(* PLC project Unnamed, Unknown Unnamed 1 *)
(* stored: creationDateTime 2024-01-22T13:26:01, modificationDateTime 2024-01-28T15:10:34 *)

PROGRAM program0
  VAR
    FactoryIOReset AT %IX100.0 : BOOL;
    Start AT %IX100.1 : BOOL := 1;
    EmergencyStop AT %IX100.2 : BOOL;
    RetroReflect0 AT %IX100.3 : BOOL;  (* Retroreflective sensors are active low which means that the signal goes from 1 to 0 when the sensor is triggered by the pallet *)
    RetroReflect1 AT %IX100.4 : BOOL;
    RetroReflect2 AT %IX100.5 : BOOL;
    RetroReflect3 AT %IX100.6 : BOOL;
    TurntableBackLimit AT %IX100.7 : BOOL;
    TurntableFrontLimit AT %IX101.0 : BOOL;
    TurntableLimit0 AT %IX101.1 : BOOL;
    TurntableLimit90 AT %IX101.2 : BOOL;
    LightArray7 AT %IX101.3 : BOOL;
    Conveyor1 AT %QX100.0 : BOOL;
    Turntable0RollPlus AT %QX100.1 : BOOL;
    Turntable0Turn AT %QX100.2 : BOOL;
    Conveyor2 AT %QX100.3 : BOOL;
  END_VAR
  VAR
    RS0 : RS;
    RS1 : RS;
    RS2 : RS;
  END_VAR
  VAR_IN_OUT
    SmallBox : BOOL;
  END_VAR
  VAR
    RS3 : RS;
    RS4 : RS;
    RS5 : RS;
    RS6 : RS;
    RS7 : RS;
    RS8 : RS;
    RS9 : RS;
  END_VAR
  VAR  (* added by the conversion: wires and edge detectors of the diagram *)
    R_TRIG1 : R_TRIG;
    R_TRIG2 : R_TRIG;
    R_TRIG3 : R_TRIG;
    R_TRIG4 : R_TRIG;
    F_TRIG5 : F_TRIG;
    R_TRIG6 : R_TRIG;
    R_TRIG7 : R_TRIG;
    R_TRIG8 : R_TRIG;
    F_TRIG9 : F_TRIG;
    R_TRIG10 : R_TRIG;
    F_TRIG11 : F_TRIG;
    R_TRIG12 : R_TRIG;
    R_TRIG13 : R_TRIG;
    R_TRIG14 : R_TRIG;
    F_TRIG15 : F_TRIG;
    R_TRIG16 : R_TRIG;
    R_TRIG17 : R_TRIG;
    F_TRIG18 : F_TRIG;
    R_TRIG19 : R_TRIG;
    R_TRIG20 : R_TRIG;
    R_TRIG21 : R_TRIG;
    R_TRIG22 : R_TRIG;
    R_TRIG23 : R_TRIG;
    R_TRIG24 : R_TRIG;
    R_TRIG25 : R_TRIG;
  END_VAR

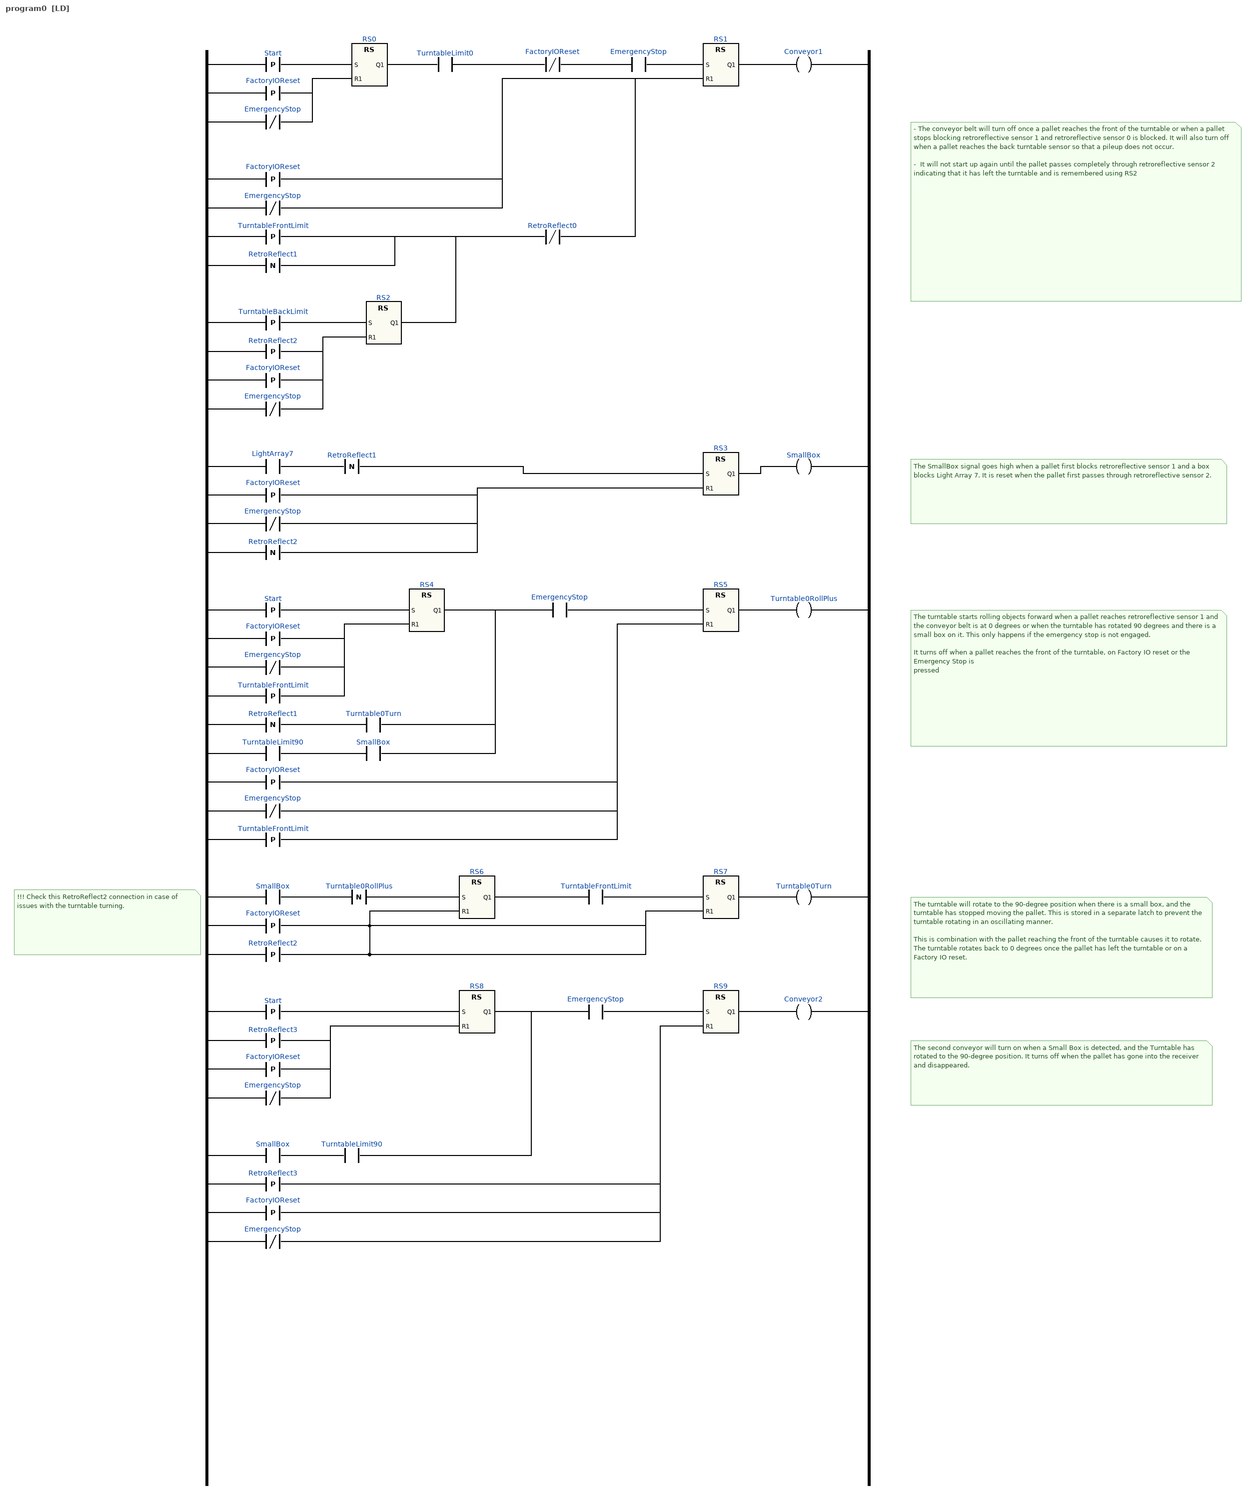
(* LD diagram, written out as Structured Text *)
R_TRIG1(CLK := Start);
R_TRIG2(CLK := FactoryIOReset);
RS0(S := R_TRIG1.Q, R1 := R_TRIG2.Q OR NOT EmergencyStop);
R_TRIG3(CLK := FactoryIOReset);
R_TRIG4(CLK := TurntableFrontLimit);
F_TRIG5(CLK := RetroReflect1);
R_TRIG6(CLK := TurntableBackLimit);
R_TRIG7(CLK := RetroReflect2);
R_TRIG8(CLK := FactoryIOReset);
RS2(S := R_TRIG6.Q, R1 := R_TRIG7.Q OR R_TRIG8.Q OR NOT EmergencyStop);
RS1(S := RS0.Q1 AND TurntableLimit0 AND NOT FactoryIOReset AND EmergencyStop, R1 := R_TRIG3.Q OR NOT EmergencyStop OR (R_TRIG4.Q OR F_TRIG5.Q OR RS2.Q1) AND NOT RetroReflect0);
Conveyor1 := RS1.Q1;
(* - The conveyor belt will turn off once a pallet reaches the front of the turntable or when a pallet stops blocking retroreflective sensor 1 and retroreflective sensor 0 is blocked. It will also turn off when a pallet reaches the back turntable sensor so that a pileup does not occur.

-  It will not start up again until the pallet passes completely through retroreflective sensor 2
indicating that it has left the turntable and is remembered using RS2 *)
(* The SmallBox signal goes high when a pallet first blocks retroreflective sensor 1 and a box blocks Light Array 7. It is reset when the pallet first passes through retroreflective sensor 2. *)
F_TRIG9(CLK := RetroReflect1);
R_TRIG10(CLK := FactoryIOReset);
F_TRIG11(CLK := RetroReflect2);
RS3(S := LightArray7 AND F_TRIG9.Q, R1 := R_TRIG10.Q OR NOT EmergencyStop OR F_TRIG11.Q);
SmallBox := RS3.Q1;
R_TRIG12(CLK := Start);
R_TRIG13(CLK := FactoryIOReset);
R_TRIG14(CLK := TurntableFrontLimit);
RS4(S := R_TRIG12.Q, R1 := R_TRIG13.Q OR NOT EmergencyStop OR R_TRIG14.Q);
F_TRIG15(CLK := RetroReflect1);
R_TRIG16(CLK := FactoryIOReset);
R_TRIG17(CLK := TurntableFrontLimit);
RS5(S := (RS4.Q1 OR F_TRIG15.Q AND Turntable0Turn OR TurntableLimit90 AND SmallBox) AND EmergencyStop, R1 := R_TRIG16.Q OR NOT EmergencyStop OR R_TRIG17.Q);
Turntable0RollPlus := RS5.Q1;
(* The turntable starts rolling objects forward when a pallet reaches retroreflective sensor 1 and the conveyor belt is at 0 degrees or when the turntable has rotated 90 degrees and there is a small box on it. This only happens if the emergency stop is not engaged.

It turns off when a pallet reaches the front of the turntable, on Factory IO reset or the Emergency Stop is 
pressed *)
(* !!! Check this RetroReflect2 connection in case of issues with the turntable turning. *)
F_TRIG18(CLK := Turntable0RollPlus);
R_TRIG19(CLK := FactoryIOReset);
R_TRIG20(CLK := RetroReflect2);
RS6(S := SmallBox AND F_TRIG18.Q, R1 := R_TRIG19.Q OR R_TRIG20.Q);
RS7(S := RS6.Q1 AND TurntableFrontLimit, R1 := R_TRIG19.Q OR R_TRIG20.Q);
Turntable0Turn := RS7.Q1;
(* The turntable will rotate to the 90-degree position when there is a small box, and the turntable has stopped moving the pallet. This is stored in a separate latch to prevent the turntable rotating in an oscillating manner. 

This is combination with the pallet reaching the front of the turntable causes it to rotate. The turntable rotates back to 0 degrees once the pallet has left the turntable or on a Factory IO reset. *)
R_TRIG21(CLK := Start);
R_TRIG22(CLK := RetroReflect3);
R_TRIG23(CLK := FactoryIOReset);
RS8(S := R_TRIG21.Q, R1 := R_TRIG22.Q OR R_TRIG23.Q OR NOT EmergencyStop);
R_TRIG24(CLK := RetroReflect3);
R_TRIG25(CLK := FactoryIOReset);
RS9(S := (RS8.Q1 OR SmallBox AND TurntableLimit90) AND EmergencyStop, R1 := R_TRIG24.Q OR R_TRIG25.Q OR NOT EmergencyStop);
Conveyor2 := RS9.Q1;
(* The second conveyor will turn on when a Small Box is detected, and the Turntable has rotated to the 90-degree position. It turns off when the pallet has gone into the receiver and disappeared. *)
END_PROGRAM

CONFIGURATION Config0
  RESOURCE Res0 ON PLC
    TASK task0(INTERVAL := T#20ms, PRIORITY := 0);
    PROGRAM instance0 WITH task0 : program0;
  END_RESOURCE
END_CONFIGURATION
